FUNCTION_BLOCK BYTE_UNION

VAR_INPUT
	Upper_Byte:			BYTE;
	Lower_Byte:			BYTE;
END_VAR

VAR_OUTPUT
	United_Word:		WORD;
END_VAR

VAR
	Aux_Word:			WORD;
END_VAR

Aux_Word:= BYTE_TO_WORD (Upper_Byte);
United_Word:= SHL (Aux_Word, 8) + Lower_Byte;

END_FUNCTION_BLOCK

(* stored: Version 1.1.0.1, ProductVersion 3.1.4024.11
   POU BYTE_UNION: Id {e7db25c2-e50c-4e4a-a487-8cf86f9ae307}, SpecialFunc None *)
